# EPICS autosave request: iocBoot/gmca_23o_ioc1/dbSave/XZ_P9_.req
%
% BURT Request File
%
% $(P)XZ:P9:  X-Y positioner #9
%

file assy.req ASSY=$(P)XZ:P9
file mtr1.req MTR1=$(P)XZ:mx9
file mtr1.req MTR1=$(P)XZ:my9
file drv1.req DRV1=$(P)XZ:X9
file drv1.req DRV1=$(P)XZ:Y9
